{attribute addProperty BoxType "KL9900-0062"}
{attribute addProperty Id "E_StopAT %I*BOOL000"}
{attribute addProperty CRC "3613501377"}
{attribute addProperty SizeInBites "0"}
{attribute addProperty SizeInBytes "0"}
TYPE Channel_D761A7C1 :
STRUCT
	{attribute addProperty Name "E_Stop"}
	E_Stop AT %I* : BOOL;
END_STRUCT
END_TYPE

(* stored: Version 1.2.0.0, ProductVersion 3.1.4024.9
   DUT Channel_D761A7C1: Id {08affed6-30d1-467b-9b4a-8c85c4aac5a2} *)
